PROGRAM PRG_TEST
VAR
    _testSuite : TcUnitContext;
END_VAR

_testSuite.Run();
_testSuite.RtcSynchronize(true, '', 60);

END_PROGRAM

(* stored: Version 1.1.0.1, ProductVersion 3.1.4024.12
   POU PRG_TEST: Id {1d4196be-6e69-0a6b-2f6d-cb981643101e}, SpecialFunc None *)
